(* IEC 61131-3 sources: Industrial-Meter-Tracking-System-Modernization/plc/structured-text, 4 files *)

(* ---- calc-delta-prg.st ---- *)
(*
    Program: CalcDelta
    Purpose:
    Analyzes pulse duration from two line sensors.

    This program calls two instances of the CalcDeltaT function block:
    - one for the input sensor
    - one for the output sensor

    The function block measures minimum and maximum pulse duration
    within configured limits.

    Note:
    This is an anonymized version of the original industrial PLC logic.
*)

PROGRAM CalcDelta
VAR
    InputSensorPulseAnalyzer  : CalcDeltaT;
    OutputSensorPulseAnalyzer : CalcDeltaT;
END_VAR

// Input sensor pulse duration analysis
InputSensorPulseAnalyzer(
    Reset    := ResetMinMax,
    Sensor   := Line_Input_Sensor,
    MIN_T_ms := 1,
    MAX_T_ms := 5000,
    MinTime  => Input_Min_Pulse_Time_ms,
    MaxTime  => Input_Max_Pulse_Time_ms
);

// Output sensor pulse duration analysis
OutputSensorPulseAnalyzer(
    Reset    := ResetMinMax,
    Sensor   := Line_Output_Sensor,
    MIN_T_ms := 1,
    MAX_T_ms := 5000,
    MinTime  => Output_Min_Pulse_Time_ms,
    MaxTime  => Output_Max_Pulse_Time_ms
);

(* ---- get-date-time-prg.st ---- *)
(*
    Program: GetDateTime
    Purpose:
    Reads PLC real-time clock, applies local time zone offset
    and splits date/time into separate variables for HMI, SCADA
    and database logic.

    Note:
    This is an anonymized representation of the original PLC logic.
*)

PROGRAM GetDateTime
VAR
    CurrentTimestampUtc : DWORD;
    CurrentDateTime     : DATE_AND_TIME;

    TimeZoneOffsetHours : DINT := 3;
    TimeZoneOffsetSec   : DINT;

    CurrentYear         : UINT;
    CurrentMonth        : UINT;
    CurrentDay          : UINT;
    CurrentHour         : UINT;
    CurrentMinute       : UINT;
    CurrentSecond       : UINT;
END_VAR

// Read PLC system time in UTC
CurrentTimestampUtc := SysTimeRtc.SysTimeRtcGet();

// Convert time zone offset from hours to seconds
TimeZoneOffsetSec := TimeZoneOffsetHours * 3600;

// Apply local time zone offset and convert timestamp to date/time
CurrentDateTime := SysTimeRtc.SysTimeRtcConvertUtcToDate(
    dwTimestampUtc := CurrentTimestampUtc + DINT_TO_DWORD(TimeZoneOffsetSec)
);

// Split date/time into separate values
CurrentYear   := CurrentDateTime.Year;
CurrentMonth  := CurrentDateTime.Month;
CurrentDay    := CurrentDateTime.Day;
CurrentHour   := CurrentDateTime.Hour;
CurrentMinute := CurrentDateTime.Minute;
CurrentSecond := CurrentDateTime.Second;

(* ---- shift-and-state-analysis.st ---- *)
(*
    Program: Shift and State Analysis
    Purpose:
    - Determines current work shift (day/night)
    - Detects shift change
    - Saves production state into history
    - Resets counters at shift boundary
    - Tracks line state changes and alarms

    Note:
    This is an anonymized and simplified version of the original logic.
*)

PROGRAM ShiftAnalysis

VAR
    PrevShift : INT;
    CurrentShift : INT;

    CurrentHour : INT;

    ResetCounters : BOOL;
    BreakDetected : BOOL;
END_VAR

// Store previous shift
PrevShift := CurrentShift;

// Determine current shift
IF (CurrentHour >= 8 AND CurrentHour < 20) THEN
    CurrentShift := 1; // Day shift
ELSE
    CurrentShift := 2; // Night shift
END_IF;

// Detect shift change
IF (PrevShift <> CurrentShift) THEN

    // Save current state to history (simplified)
    SaveToHistory(
        Shift := PrevShift,
        Timestamp := CurrentTime,
        Status := LineStatus
    );

    // Reset production counters
    ResetCounters := TRUE;

END_IF;

// Time validation (simplified)
IF (MaterialAnalysisTime < 1) THEN
    MaterialAnalysisTime := 1;
END_IF;

IF (WorkAnalysisTime <= MaterialAnalysisTime) THEN
    WorkAnalysisTime := MaterialAnalysisTime + 1;
END_IF;

// Decode status word
DecodeStatusWord(
    StatusWord := LineStatus,
    BreakSignal => BreakDetected
);

// If break event detected — log it
IF (BreakDetected) THEN
    SaveBreakEvent(
        AlarmCode := AlarmCodeValue,
        Timestamp := CurrentTime
    );
END_IF;

(* ---- transfer-to-db-prg.st ---- *)
(*
    Program: Transfer_To_DB
    Purpose:
    Prepares historical production records for transfer from PLC to SCADA / SQL database.

    Transfer handshake logic:
    0 - PLC is ready to prepare next record
    1 - PLC prepared a record, server can read it
    2 - server confirmed that the record was read

    Note:
    This is an anonymized and simplified version of the original PLC logic.
*)

PROGRAM Transfer_To_DB
VAR
    RecordReadyForTransfer : BOOL;
    TransferDelay          : TON;

    TransferState          : INT;  // 0 = ready, 1 = data prepared, 2 = server confirmed
    HistoryIndex           : INT;
    LastHistoryIndex       : INT;

    CurrentShift           : INT;
    CurrentHour            : INT;
END_VAR

// Determine current shift
IF (CurrentHour >= 8 AND CurrentHour < 20) THEN
    CurrentShift := 1; // Day shift
ELSE
    CurrentShift := 2; // Night shift
END_IF;

// If server confirmed that data was read
IF (TransferState = 2) THEN

    TransferState := 0; // Ready for next record

    History[HistoryIndex].NotTransferred := FALSE;

    HistoryIndex := HistoryIndex + 1;

    IF (HistoryIndex > LastHistoryIndex) THEN
        HistoryIndex := LastHistoryIndex;
    END_IF;

END_IF;

// Prepare next not-transferred record
IF (TransferState = 0) THEN

    IF (History[HistoryIndex].NotTransferred = TRUE) THEN

        // Copy historical data to transfer buffer
        TransferBuffer.Year          := History[HistoryIndex].Year;
        TransferBuffer.Month         := History[HistoryIndex].Month;
        TransferBuffer.Day           := History[HistoryIndex].Day;
        TransferBuffer.Hour          := History[HistoryIndex].Hour;
        TransferBuffer.Minute        := History[HistoryIndex].Minute;
        TransferBuffer.Second        := History[HistoryIndex].Second;

        TransferBuffer.InputCounter  := History[HistoryIndex].InputCounter;
        TransferBuffer.OutputCounter := History[HistoryIndex].OutputCounter;
        TransferBuffer.FalseCounter  := History[HistoryIndex].FalseCounter;

        TransferBuffer.OrderNumber   := History[HistoryIndex].OrderNumber;
        TransferBuffer.StatusWord    := History[HistoryIndex].StatusWord;
        TransferBuffer.SetupType     := History[HistoryIndex].SetupType;
        TransferBuffer.UserNumber    := History[HistoryIndex].UserNumber;
        TransferBuffer.ShiftNumber   := History[HistoryIndex].ShiftNumber;

        // Delay before setting ready flag
        TransferDelay(
            IN := History[HistoryIndex].NotTransferred,
            PT := T#2S
        );

        IF (TransferDelay.Q) THEN
            TransferState := 1; // Data prepared, server can read it
            TransferDelay(IN := FALSE);
        END_IF;

    ELSE

        // Skip already transferred records
        HistoryIndex := HistoryIndex + 1;

        IF (HistoryIndex > LastHistoryIndex) THEN
            HistoryIndex := LastHistoryIndex;
        END_IF;

    END_IF;

END_IF;

// Reset Modbus reset command after transfer cycle
ModbusResetCommand := 0;
